FUNCTION_BLOCK GenericQueue
VAR_INPUT CONSTANT
	dataSize : UDINT; //no functionaility, only to force input a type for readability
END_VAR
VAR //pointers = 8 byte integers
	elements : FB_BA_DynamicArray := (uiEntrySize := SIZEOF(POINTER TO UnionQ), uiMinExpCount := GVL.initArraySize);
	length : USINT := 0;
END_VAR

METHOD clear : BOOL
VAR_INPUT
END_VAR
elements.Reset();
length := 0;
END_METHOD

METHOD contains : BOOL
VAR_INPUT
	value : UnionQ;
END_VAR
VAR_INST
	i : INT;
END_VAR
IF length = 0 THEN
	contains := FALSE;
	RETURN;
END_IF

FOR i:=0 TO length-1 BY 1 DO
	IF MEMCMP(get(i), ADR(value), SIZEOF(UnionQ)) = 0 THEN
		contains := TRUE;
		RETURN;
	END_IF
END_FOR
contains := FALSE;
END_METHOD

METHOD get : POINTER TO UnionQ
VAR_INPUT
	i : INT;
END_VAR
IF length = 0 OR i < 0 OR i >= length THEN
	get := 0;
ELSE
	elements.GetEntry(diIndex := i, pResultEntry := ADR(get));
END_IF
END_METHOD

METHOD isEmpty : BOOL
VAR_INPUT
END_VAR
isEmpty := length = 0;
END_METHOD

METHOD poll : POINTER TO UnionQ
VAR
	temp : POINTER TO UnionQ;
	i : INT;
END_VAR
poll := get(i := 0);

IF length > 0 THEN
	elements.RemoveEntry(diIndex := 0);
	length := length - 1;
END_IF
END_METHOD

METHOD push : BOOL
VAR_INPUT
	value : POINTER TO UnionQ;
END_VAR
elements.AddEntry(pEntry := ADR(value));
length := length + 1;
END_METHOD

METHOD set : BOOL
VAR_INPUT
	i : INT;
	value : POINTER TO UnionQ;
END_VAR
IF i > 0 AND i < length THEN
	elements.SetEntry(i, ADR(value));
	set := TRUE;
END_IF
END_METHOD

METHOD size : USINT
size := length;
END_METHOD

END_FUNCTION_BLOCK

(* stored: Version 1.1.0.1, ProductVersion 3.1.4024.11
   POU GenericQueue: Id {e7bca9f7-e2c1-41e8-9e98-f6a9133845a3}, SpecialFunc None
   Method clear: Id {d720abaa-113a-463a-8cb1-0f64b55d1c80}
   Method contains: Id {417b1983-67bb-416d-bd55-13a0fe5ca3b3}
   Method get: Id {0b2fa2c1-3d44-4975-9ce0-c9473517d753}
   Method isEmpty: Id {31d66a9c-50a3-4fcd-850e-6bdefaaf28fd}
   Method poll: Id {1f7ff33a-a91e-4842-a8da-4414a3544d77}
   Method push: Id {dce80655-efb8-426b-a022-f478e223b154}
   Method set: Id {3f3298cf-ea2c-441a-945c-342cf9c7de98}
   Method size: Id {0d97d89b-4bee-4ed5-bc09-af7514b6de18} *)
